(*
RMatrix : 3D Rotation Matrix
======================

Overview
----------------------

This class represents a 3x3 matrix used to represent a rotation.

See: `https://en.wikipedia.org/wiki/Rotation_matrix`__

You can think of the RMatrix as representing the orientation of  *child* coordinate system inside a *parent* coordinate system. 
Each column vector of the RMatrix is essentially a unit vector (X, Y, or Z) of the child coordinate system projected into the parent coordinate system.
Premultiplication with this matrix transforms vectors and other rotations out of the child coordinate system and into the parent coordinate system. 
Reversing the RMatrix simply reverses the roles (parent/child) of the coordinate system and allows transformations in the other direction.
*)
{attribute 'reflection'}
FUNCTION_BLOCK RMatrix EXTENDS StaticMatrix
VAR_INPUT
END_VAR
VAR_OUTPUT
END_VAR
VAR
	Data : ARRAY[0..cRows*cCols-1] OF LREAL;
	ReversedAccessor_ : TransposeMatrixAccessor;//reinitialize every use (via property) because := copying will destroy the pointer
END_VAR
VAR CONSTANT
	cRows : UINT := 3;
	cCols : UINT := 3;
END_VAR

METHOD PROTECTED BuildFromUnitVectors
VAR_INPUT
	X : REFERENCE TO Vector3;
	Y : REFERENCE TO Vector3;
	Z : REFERENCE TO Vector3;
END_VAR
FillFromAt(X,0,0);
FillFromAt(Y,0,1);
FillFromAt(Z,0,2);
END_METHOD

METHOD PUBLIC Clear
VAR_INPUT
END_VAR
FillTrapezoidal(1,0,0);
END_METHOD

METHOD FB_init : BOOL
VAR_INPUT
	bInitRetains : BOOL; // if TRUE, the retain variables are initialized (warm start / cold start)
	bInCopyCode : BOOL;  // if TRUE, the instance afterwards gets moved into the copy code (online change)
END_VAR
Init_(cRows,cCols);
Clear();
END_METHOD

//Returns a ZYX tait-Bryan angle sequence that represents this rotation matrix
METHOD PUBLIC GetAngleSequence : TaitBryanAngleOrientation
VAR_INPUT
END_VAR
GetAngleSequence.Sequence := TaitBryanAngleSequence.ZYX;
IF GetRC(0,0) = 0 OR GetRC(1,0) = 0 THEN
	GetAngleSequence.RzRad := 0;
	GetAngleSequence.RyRad := PI/2;
	GetAngleSequence.RxRad := ATAN2(GetRC(0,1),GetRC(1,1));
ELSE
	GetAngleSequence.RzRad := ATAN2(GetRC(1,0),GETRC(0,0));
	GetAngleSequence.RyRad := ATAN2(-1*GetRC(2,0),SQRT(GetRC(0,0)*GetRC(0,0) + GetRC(1,0)*GetRC(1,0)));
	GetAngleSequence.RxRad := ATAN2(GetRC(2,1),GetRC(2,2));
END_IF
END_METHOD

//Gets the value of the element in this matrix at the supplied location as if the elements were stored in a 1D row-major array
//:Prerequisites:
// - I < Rows*Cols
// - Matrix is not empty
//If the supplied index is out of bounds the value 0 is returned and a warning is generated in the Error List
METHOD PUBLIC GetI : LREAL//The value of the element at the specified index, or 0 if an invalid index is supplied
VAR_INPUT
	I : UINT;//The index of the element which should have its value returned
END_VAR
IF I >= Length THEN
	GetI := 0.0;
	LogWarning('%s: Attempted I access of out-of-bounds Matrix data');
ELSE
	GetI := Data[I];
END_IF
END_METHOD

METHOD PUBLIC GetReversed : RMatrix
VAR_INPUT
END_VAR
GetReversed := THIS^;
GetReversed.Reverse();
END_METHOD

METHOD PUBLIC GetRotatedRMatrix : RMatrix;
VAR_INPUT
	M_R : REFERENCE TO RMatrix;
END_VAR
RotateRMatrix(M_R,GetRotatedRMatrix);
END_METHOD

METHOD PUBLIC GetRotatedRMatrixReverse : RMatrix;
VAR_INPUT
	M_R : REFERENCE TO RMatrix;
END_VAR
RotateRMatrixReverse(M_R,GetRotatedRMatrixReverse);
END_METHOD

METHOD PUBLIC GetRotatedVector3 : Vector3
VAR_INPUT
	M_V : Vector3;
END_VAR
RotateVector3(M_V,GetRotatedVector3);
END_METHOD

METHOD PUBLIC GetRotatedVector3Reverse : Vector3
VAR_INPUT
	M_V : Vector3;
END_VAR
RotateVector3Reverse(M_V,GetRotatedVector3Reverse);
END_METHOD

METHOD PUBLIC Reverse
VAR_INPUT
END_VAR
Matrix_TransposeSquare(THIS^);
END_METHOD

PROPERTY PROTECTED ReversedAccessor : REFERENCE TO Matrix
GET
ReversedAccessor_.Init(THIS^);
ReversedAccessor REF= ReversedAccessor_;
END_GET
END_PROPERTY

//Equivalent to Matrix Operation 'THIS := M_R * THIS'
METHOD PUBLIC RotateBy
VAR_INPUT
	M_R : REFERENCE TO RMatrix;
END_VAR
VAR
	Temp : RMatrix := THIS^;
END_VAR
M_R.RotateRMatrix(Temp,THIS^);
END_METHOD

//Equivalent to Matrix Operation 'THIS := M_R * THIS'
METHOD PUBLIC RotateByReverse
VAR_INPUT
	M_R : REFERENCE TO RMatrix;
END_VAR
VAR
	Temp : RMatrix := THIS^;
END_VAR
M_R.RotateRMatrixReverse(Temp,THIS^);
END_METHOD

METHOD PUBLIC RotateRMatrix
VAR_INPUT
	R_From : REFERENCE TO RMatrix;
	R_To : REFERENCE TO RMatrix;
END_VAR
Matrix_Product(THIS^,R_From,R_To);
END_METHOD

METHOD PUBLIC RotateRMatrixReverse
VAR_INPUT
	R_From : REFERENCE TO RMatrix;
	R_To : REFERENCE TO RMatrix;
END_VAR
Matrix_Product(ReversedAccessor,R_From,R_To);
END_METHOD

METHOD PUBLIC RotateVector3
VAR_INPUT
	V_From : REFERENCE TO Vector3;
	V_To : REFERENCE TO Vector3;
END_VAR
Matrix_Product(THIS^,V_From,V_To);
END_METHOD

METHOD PUBLIC RotateVector3Reverse
VAR_INPUT
	V_From : REFERENCE TO Vector3;
	V_To : REFERENCE TO Vector3;
END_VAR
Matrix_Product(ReversedAccessor,V_From,V_To);
END_METHOD

METHOD PUBLIC SetFromAngle
VAR_INPUT
	Angle : LREAL;//radians
	Dimension : Dimension;//0-2
END_VAR
VAR
	SM : ShrunkMatrixAccessor;
	Sign : LREAL;
	
END_VAR
FillTrapezoidal(1,0,0);
Sign := INT_TO_LREAL(((UINT_TO_INT(Dimension) MOD 2)*2)-1);
SM := GetShrunkMatrixAccessor(Dimension,Dimension);
SM.FillTrapezoidal(COS(Angle),Sign*SIN(Angle),-1*Sign*SIN(Angle));
END_METHOD

//Intrinsic Rotations
METHOD PUBLIC SetFromAngleSequence
VAR_INPUT
END_VAR
VAR_IN_OUT
	Angles : ARRAY [*] OF LREAL;
	Dimensions : ARRAY [*] OF Dimension;
END_VAR
VAR
	I : DINT;
	N : DINT;
	RTemp : RMatrix;
END_VAR
N := MIN(UPPER_BOUND(Angles,1) - LOWER_BOUND(Angles,1),UPPER_BOUND(Dimensions,1) - LOWER_BOUND(Dimensions,1))+1;
FillTrapezoidal(1,0,0);
FOR I := N-1 TO 0 BY -1 DO
	RTemp.SetFromAngle(Angles[LOWER_BOUND(Angles,1)+I],Dimensions[LOWER_BOUND(Dimensions,1)+I]);
	RotateBy(RTemp);
END_FOR
END_METHOD

METHOD PUBLIC SetFromVectorsXY : BOOL
VAR_INPUT
	X : VEctor3;//make a copy so we can nromalize
	Y : Vector3;//make a copy so we can normalize
END_VAR
VAR
	Z : Vector3;
END_VAR
IF X.GetVector3DotProduct(Y) <> 0 THEN
	LogWarning('%s: attempt to build RMatrix from non-perpendicular vectors');
	SetFromVectorsXY := FALSE;
	RETURN;
END_IF
SetFromVectorsXY := TRUE;
X.Normalize();
Y.Normalize();
Z.SetAsCrossProduct(X,Y);
BuildFromUnitVectors(X,Y,Z);
END_METHOD

METHOD PUBLIC SetFromVectorsXZ : BOOL
VAR_INPUT
	X : VEctor3;//make a copy so we can nromalize
	Z : Vector3;//make a copy so we can normalize
END_VAR
VAR
	Y : Vector3;
END_VAR
IF X.GetVector3DotProduct(Z) <> 0 THEN
	LogWarning('%s: attempt to build RMatrix from non-perpendicular vectors');
	SetFromVectorsXZ := FALSE;
	RETURN;
END_IF
SetFromVectorsXZ := TRUE;
X.Normalize();
Z.Normalize();
Y.SetAsCrossProduct(Z,X);
BuildFromUnitVectors(X,Y,Z);
END_METHOD

METHOD PUBLIC SetFromVectorsYZ : BOOL
VAR_INPUT
	Y : VEctor3;//make a copy so we can nromalize
	Z : Vector3;//make a copy so we can normalize
END_VAR
VAR
	X : Vector3;
END_VAR
IF Y.GetVector3DotProduct(Z) <> 0 THEN
	LogWarning('%s: attempt to build RMatrix from non-perpendicular vectors');
	SetFromVectorsYZ := FALSE;
	RETURN;
END_IF
SetFromVectorsYZ := TRUE;
Y.Normalize();
Z.Normalize();
X.SetAsCrossProduct(Y,Z);
BuildFromUnitVectors(X,Y,Z);
END_METHOD

//Sets the element specified by the supplied index to the suppleid value, assuming the data of the matrix is stored in a 1D row-major array
//:Prerequisites: - I < Rows*Cols
METHOD PUBLIC SetI : BOOL//TRUE if the specified index is valid and the data is copied. FLASE otherwise
VAR_INPUT
	I : UINT;//The index specifying which element should be modified
	Val : LREAL;//The value copied to the corresponding element
END_VAR
IF I >= Length THEN
	SetI := FALSE;
	LogWarning('%s: Attempt to set data using I access when I is out of bounds');
ELSE
	SetI := TRUE;
	Data[I] := Val;
END_IF
END_METHOD

END_FUNCTION_BLOCK

(* stored: Version 1.1.0.1, ProductVersion 3.1.4024.9
   POU RMatrix: Id {9bc066e0-5060-4767-b54e-f3a680b769d5}, SpecialFunc None
   Folder Getters: Id {80c3ef77-8bb8-42f3-a586-d0dc3a38b4a1}
   Folder Helpers: Id {ccf67a90-57bb-4b16-8e9c-6f84260aaabf}
   Folder Modifiers: Id {0f6c6206-349d-4c60-ae1d-9d55fe206d70}
   Folder Overrides: Id {af5c3a94-d6f7-4c2c-800b-35fdadbd3f54}
   Folder Properties: Id {a664b485-ddbc-0c87-0f0c-cf9c70fb7180}
   Folder Protected: Id {d4a9f165-5d92-0d5d-15d3-89558c4f1a79}
   Folder Setters: Id {f7cadddc-161a-48bc-a94b-177606fba9de}
   Method BuildFromUnitVectors: Id {a254d824-c923-02fe-3444-221d65b9dea3}
   Method Clear: Id {027f050f-4f77-4aeb-a0e0-39072a4e57ce}
   Method FB_init: Id {26ea4d11-e89f-43a1-af7e-c6b796c00b93}
   Method GetAngleSequence: Id {ae6629b9-f5bd-02fe-28d9-e01a4b8ce654}
   Method GetI: Id {015a9ab6-358d-413c-971b-ae0068470b6d}
   Method GetReversed: Id {92a4b7bf-86be-4bea-af13-ea62374ec0d7}
   Method GetRotatedRMatrix: Id {af9e57ab-1242-4d2a-bea1-322f456421a1}
   Method GetRotatedRMatrixReverse: Id {939de2bb-a599-0eff-3c8c-61d7b368e042}
   Method GetRotatedVector3: Id {98fbe1a3-cb09-4e8d-af7b-b0032dd8f73e}
   Method GetRotatedVector3Reverse: Id {eb5c710c-f386-012c-16fa-2069a4fde340}
   Method Reverse: Id {c0867d18-4c42-4215-9a97-1688df15e7cb}
   Property ReversedAccessor: Id {7e5b2534-b7ec-07df-36e1-807beb6e44ec}
   Get Get: Id {661a0efc-82cb-0675-2029-4ff3a2ffa1f1}
   Method RotateBy: Id {c7db5993-9ae0-46f4-b208-76cc11903f65}
   Method RotateByReverse: Id {7bfc985b-ffb9-0936-36f2-d34bd9ff7817}
   Method RotateRMatrix: Id {94514cca-3495-4305-a7b1-caebc38d65fe}
   Method RotateRMatrixReverse: Id {bfdecbfc-95fe-03b6-2db4-7ab7c8d3a901}
   Method RotateVector3: Id {a1d2c87d-b7d5-4de7-bf30-62e9d26671c1}
   Method RotateVector3Reverse: Id {1ef31973-3fba-0dc5-1845-e8f8eb51537f}
   Method SetFromAngle: Id {a4f2a576-ecea-4d2e-ba8e-23d82bdf48d3}
   Method SetFromAngleSequence: Id {1d13de46-a9bc-418e-b26e-cffe204950b3}
   Method SetFromVectorsXY: Id {67916213-bf7a-0008-2fb8-686aa9434c37}
   Method SetFromVectorsXZ: Id {017ae7e6-4063-04a5-1826-1e88b3a28ef6}
   Method SetFromVectorsYZ: Id {489e46e9-01d1-003d-18db-ab7410c00b7f}
   Method SetI: Id {01d3b92f-75e1-4b02-848a-872990a093d9} *)
